
// ===== library types =====

TYPE "UDT_STRUCTANYPTR"
TITLE = 'DISSASEMBLED ANYPOINTER'
   STRUCT
      S7Code : Byte;
      DataType : Byte;
      Length : Int;
      DBNumber : Int;
      MemoryArea : Byte;
      ByteAddressMSB : Byte;
      ByteAddressLSB : Word;
   END_STRUCT;
END_TYPE

// ===== library: MasterCopy "Unixtime" =====

FUNCTION "Unixtime" : Void   // FC114, SCL
{ S7_Optimized_Access := 'FALSE' }
VERSION : 0.1
// ported by Groschke to TIA V13
BEGIN
   #leapyears := 0;
   #days_from_1970 := 0;

   // days of current month without leap day

   #days_from_BeginOfYear[0] := 0;
   #days_from_BeginOfYear[1] := 31;
   #days_from_BeginOfYear[2] := 59;
   #days_from_BeginOfYear[3] := 90;
   #days_from_BeginOfYear[4] := 120;
   #days_from_BeginOfYear[5] := 151;
   #days_from_BeginOfYear[6] := 181;
   #days_from_BeginOfYear[7] := 212;
   #days_from_BeginOfYear[8] := 243;
   #days_from_BeginOfYear[9] := 273;
   #days_from_BeginOfYear[10] := 304;
   #days_from_BeginOfYear[11] := 334;


   // read system time
   #sfc1_ret_val := RD_SYS_T(OUT => #CDT_systemtime);
   #year := BCD16_TO_INT(#systemtime.year_CDT) + 2000;
   #month := BCD16_TO_INT(#systemtime.month_CDT);
   #day := BCD16_TO_INT(#systemtime.day_CDT);
   #hour := BCD16_TO_INT(#systemtime.hour_CDT);
   #minute := BCD16_TO_INT(#systemtime.minute_CDT);
   #second := BCD16_TO_INT(#systemtime.second_CDT);


   // sum of leap years since 1979 (without current leap year)
   #leapyears := ((#year - 1) - 1968) / 4
   - ((#year - 1) - 1900) / 100
   + ((#year - 1) - 1600) / 400;


   #days_from_1970 := (#year - 1970) * 365 + #leapyears
   + #days_from_BeginOfYear[#month] + #day - 1;

   IF ((#month > 2) AND ((#year MOD 4 = 0) AND ((#year MOD 100 <> 0) OR (#year MOD 400 = 0)))) THEN
       #days_from_1970 := #days_from_1970 + 1; // + leap day, if year is leap year
   END_IF;

   // OUTPUT in s
   #l_unixtime := #second + 60 * (#minute + 60 * (#hour + 24 * #days_from_1970));


   // if error return 0
   IF #sfc1_ret_val <> 0 THEN
       #Unixtime := 0;
   ELSE
       #Unixtime := DINT_TO_DWORD(#l_unixtime);
   END_IF;
END_FUNCTION

// ===== library: MasterCopy "mqttExample" =====

FUNCTION_BLOCK "mqttExample"   // FB70, SCL
TITLE = 'MQTT Example Application'
{ S7_Optimized_Access := 'FALSE' }
AUTHOR : Brand
VERSION : 1.0
BEGIN
END_FUNCTION_BLOCK

// ===== library: MasterCopy "mqttRuntime" =====

FUNCTION_BLOCK "mqttRuntime"   // FB102, SCL
TITLE = 'Runtimercounter'
{ S7_Optimized_Access := 'FALSE' }
AUTHOR : Groschke
VERSION : 1.0
// ported by Groschke to TIA V13
BEGIN

   IF #IN AND NOT #FP_IN THEN
     #last := 0;
     #FP_IN := true;
   END_IF;

   IF NOT #IN AND #FP_IN THEN
     #FP_IN := false;
   END_IF;


   IF #IN AND NOT #RES THEN
     #now := DWORD_TO_DINT("Unixtime"());
     IF #last = 0 THEN
       #last := #now;
       GOTO Out;
     ELSE
       #run := #run + (#now - #last);
       #last := #now;
     END_IF;

   END_IF;

   IF #IN AND #RES THEN
     #run := 0;
     #now := 0;
     #last := 0;
   ELSIF NOT #IN AND #RES THEN
     #run := 0;
     #now := 0;
     #last := 0;
   END_IF;

   IF #run >= 2073600 THEN // avoid overflow of time typ 
     #run := 0;
   END_IF;

   Out:
   #RTIME := DINT_TO_TIME(#run * 1000);
END_FUNCTION_BLOCK

// ===== library: MasterCopy "mqttGlobals" =====

DATA_BLOCK "mqttGlobals"   // DB111
TITLE = 'MQTT CONSTANTS'
{ S7_Optimized_Access := 'FALSE' }
AUTHOR : Brand
VERSION : 0.1
   VAR
      MQTT_KEEPALIVE : Time;
      MQTT_SOCKET_TIMEOUT : Time;
      TCP_RECVBUFFERSIZE : Int;
      TCP_MAXRECVSIZE : Int;
      TCP_SENDBUFFERSIZE : Int;
      TCP_TIMEOUT : Time;
      MQTT_STATE_DISCONNECT : Int;
      MQTT_STATE_DISCONNECTING : Int;
      MQTT_CONNECTION_TIMEOUT : Int;
      MQTT_CONNECTION_LOST : Int;
      MQTT_CONNECT_FAILED : Int;
      MQTT_DISCONNECTED : Int;
      MQTT_CONNECTING : Int;
      MQTT_CONNECTED : Int;
      MQTT_CONN_ACCEPTED : Int;
      MQTT_CONN_BAD_PROTOCOL : Int;
      MQTT_CONN_BAD_CLIENT_ID : Int;
      MQTT_CONN_SRVUNAVAIL : Int;
      MQTT_CONN_BAD_CREDEN : Int;
      MQTT_CONN_UNAUTHORIZED : Int;
      MQTTCONNECT : Int;
      MQTTCONNACK : Int;
      MQTTPUBLISH : Int;
      MQTTPUBACK : Int;
      MQTTPUBREC : Int;
      MQTTPUBREL : Int;
      MQTTPUBCOMP : Int;
      MQTTSUBSCRIBE : Int;
      MQTTSUBACK : Int;
      MQTTUNSUBSCRIBE : Int;
      MQTTUNSUBACK : Int;
      MQTTPINGREQ : Int;
      MQTTPINGRESP : Int;
      MQTTDISCONNECT : Int;
      MQTTReserved : Int;
      MQTTQOS0 : Int;
      MQTTQOS1 : Int;
      MQTTQOS2 : Int;
   END_VAR
BEGIN
END_DATA_BLOCK

// ===== library: MasterCopy "mqttGetNextMessageID" =====

FUNCTION "mqttGetNextMessageID" : Void   // FC103, SCL
TITLE = 'MQTT Message ID Generator'
{ S7_Optimized_Access := 'FALSE' }
AUTHOR : Brand
VERSION : 1.0
BEGIN
     "mqttData".nextMsgId := "mqttData".nextMsgId + 1;

     IF ("mqttData".nextMsgId <= 0) THEN
       "mqttData".nextMsgId := 1;
     END_IF;

     #mqttGetNextMessageID := "mqttData".nextMsgId;
END_FUNCTION

// ===== library: MasterCopy "mqttCONNECT" =====

FUNCTION "mqttCONNECT" : Void   // FC101, SCL
TITLE = 'MQTT Connect Function'
{ S7_Optimized_Access := 'FALSE' }
AUTHOR : Brand
VERSION : 1.0
// ported by Groschke to TIA V13
BEGIN
END_FUNCTION

// ===== library: MasterCopy "mqttSimpleCONNECT" =====

FUNCTION "mqttSimpleCONNECT" : Void   // FC109, SCL
TITLE = 'MQTT Connect Function (basic parameters)'
{ S7_Optimized_Access := 'FALSE' }
AUTHOR : Brand
VERSION : 1.0
// ported by Groschke to TIA V13
BEGIN
     #l_clientID := #clientID;
     #l_cleanSession := #cleanSession;

     "mqttCONNECT"(clientID := #l_clientID,
                   withUsername := false,
                   withPassword := false,
                   cleanSession := #l_cleanSession,
                   withWill := false,
                   willQos := 0,
                   willRetain := 0,
                   willTopic := '',
                   willPayload := NULL,
                   willPayloadLength := 0,
                   username := '',
                   password := '');
END_FUNCTION

// ===== library: MasterCopy "mqttDISCONNECT" =====

FUNCTION "mqttDISCONNECT" : Void   // FC102, SCL
TITLE = 'MQTT Disconnect Function'
{ S7_Optimized_Access := 'FALSE' }
AUTHOR : Brand
VERSION : 1.0
// ported by Groschke to TIA V13
BEGIN
     "mqttData".buffer[0] := INT_TO_BYTE("mqttGlobals".MQTTDISCONNECT);
     "mqttData".buffer[1] := 0;
     "mqttSendTCP"(offset := 0,
                   size := 2);
     "mqttData".lastOutActivity := "mqttData".runTime;
     "mqttData"._state := "mqttGlobals".MQTT_DISCONNECTED;
END_FUNCTION

// ===== library: MasterCopy "mqttSUBSCRIBE" =====

FUNCTION "mqttSUBSCRIBE" : Void   // FC110, SCL
TITLE = 'MQTT Subscribe Function'
{ S7_Optimized_Access := 'FALSE' }
AUTHOR : Brand
VERSION : 1.0
// ported by Groschke to TIA V13
BEGIN

   // if there's no MQTT connection return
   IF "mqttData"._state = "mqttGlobals".MQTT_DISCONNECTED THEN
     RETURN;
   END_IF;

   #l_topic := #topic;

   // check if topic is not longer than 119 bytes
   IF (128 < (9 + LEN(#l_topic))) THEN
     RETURN;
   END_IF;

   #length := 5;

   // set message ID
   #thisMessageID := "mqttGetNextMessageID"();
   "mqttData".buffer[#length] := DWORD_TO_BYTE(SHR(IN := INT_TO_DWORD(#thisMessageID), N := 8));
   #length := #length + 1;
   "mqttData".buffer[#length] := INT_TO_BYTE(#thisMessageID) AND B#16#FF;
   #length := #length + 1;

   // set topic                
   #length := "mqttWriteString"(str := #l_topic, pos := #length);

   // set topic qos
   "mqttData".buffer[#length] := INT_TO_BYTE(#topicQos);
   #length := #length + 1;

   // write header and send message
   "mqttWrite"(header := INT_TO_BYTE("mqttGlobals".MQTTSUBSCRIBE),
               length := #length - 5);
END_FUNCTION

// ===== library: MasterCopy "mqttUNSUBSCRIBE" =====

FUNCTION "mqttUNSUBSCRIBE" : Void   // FC111, SCL
TITLE = 'MQTT Unsubscribe Function'
{ S7_Optimized_Access := 'FALSE' }
AUTHOR : Brand
VERSION : 1.0
BEGIN

   // if there's no MQTT connection return
   IF "mqttData"._state = "mqttGlobals".MQTT_DISCONNECTED THEN
     RETURN;
   END_IF;

   #l_topic := #topic;

   // check if topic is not longer than 119 bytes
   IF (128 < (9 + LEN(#l_topic))) THEN
     RETURN;
   END_IF;

   #length := 5;

   // set message ID
   #thisMessageID := "mqttGetNextMessageID"();
   "mqttData".buffer[#length] := DWORD_TO_BYTE(SHR(IN := INT_TO_DWORD(#thisMessageID), N := 8));
   #length := #length + 1;
   "mqttData".buffer[#length] := INT_TO_BYTE(#thisMessageID) AND B#16#FF;
   #length := #length + 1;

   // set topic        
   #length := "mqttWriteString"(str := #l_topic, pos := #length);

   #fixedHeader := INT_TO_BYTE("mqttGlobals".MQTTUNSUBSCRIBE);
   // Set Header Flags for duplicates, qos level and retain
   #fixedHeader := #fixedHeader OR SHL(IN := BOOL_TO_BYTE(true), N := 1);

   // write header and send message
   "mqttWrite"(header := #fixedHeader,
               length := #length - 5);
END_FUNCTION

// ===== library: MasterCopy "mqttPUBLISH" =====

FUNCTION "mqttPUBLISH" : Void   // FC105, SCL
TITLE = MQTT Publish Function
{ S7_Optimized_Access := 'FALSE' }
AUTHOR : Brand
VERSION : 1.0
// ported by Groschke to TIA V13
BEGIN
   // set return value (message ID) to 0
   #mqttPUBLISH := 0;

   // if there's no MQTT connection return an error code
   IF "mqttData"._state = "mqttGlobals".MQTT_DISCONNECTED THEN
     #mqttPUBLISH := -1;
     RETURN;
   END_IF;

   // Fixed header, byte 1
   // +--------+---+-----+---+---+----------+-----+-----+--------+
   // |bit     | 7 |  6  | 5 | 4 |     3    |  2  |  1  |    0   |
   // +--------+---+-----+---+---+----------+-----+-----+--------+
   // |byte 1  | Message Type(3) | DUP Flag | QoS level | RETAIN |
   // +--------+-----------------+----------+-----------+--------+

   // set package type in header
   #fixedHeader := INT_TO_BYTE("mqttGlobals".MQTTPUBLISH);
   // Set Header Flags for duplicates, qos level and retain
   #fixedHeader := #fixedHeader OR SHL(IN := BOOL_TO_BYTE(#duplicate), N := 3) OR SHL(IN := INT_TO_BYTE(#qos), N := 1) OR BOOL_TO_BYTE(#retain);

   // Fixed header, byte 2
   // +--------+---+---+---+---+---+---+---+---+
   // |bit     | 7 | 6 | 5 | 4 | 3 | 2 | 1 | 0 |
   // +--------+---+---+---+---+---+---+---+---+
   // |bytes 2..4|   Remaining Length          |
   // +--------+-------------------------------+

   // Variable header, topic
   // +--------+---+---+---+---+---+---+---+---+
   // |bit     | 7 | 6 | 5 | 4 | 3 | 2 | 1 | 0 |
   // +--------+---+---+---+---+---+---+---+---+
   // |byte    |           Topic length MSB    |
   // +~~~~~~~~|~~~~~~~~~~~~~~~~~~~~~~~~~~~~~~~+
   // |byte    |           Topic length LSB    |
   // +~~~~~~~~|~~~~~~~~~~~~~~~~~~~~~~~~~~~~~~~+
   // +--------+---+---+---+---+---+---+---+---+
   // |bit     | 7 | 6 | 5 | 4 | 3 | 2 | 1 | 0 |
   // +--------+---+---+---+---+---+---+---+---+
   // |bytes    |           Topic              |
   // +~~~~~~~~|~~~~~~~~~~~~~~~~~~~~~~~~~~~~~~~+

   // point to buffer area in front of fixed header (5 bytes)
   // copy topic to buffer
   #holdstring := #topic;
   #length := 5;

   #length := "mqttWriteString"(str := #holdstring, pos := #length);

   // MessageID  
   // Variable header, byte 9
   // +--------+---+---+---+---+---+---+---+---+
   // |bit     | 7 | 6 | 5 | 4 | 3 | 2 | 1 | 0 |
   // +--------+---+---+---+---+---+---+---+---+           
   // |byte    |       Message ID LSB (0)      |
   // +--------+-------------------------------+ 
   // |byte    |       Message ID LSB (10)     |
   // +--------+-------------------------------+

   // set MessageID if qos level 1 or 2
   IF (#qos = "mqttGlobals".MQTTQOS1) OR (#qos = "mqttGlobals".MQTTQOS2) THEN
     IF #messageid > 0 THEN
       #thisMessageID := #messageid;
     ELSE
       #thisMessageID := "mqttGetNextMessageID"();
     END_IF;

     // insert message ID
     "mqttData".buffer[#length] := DWORD_TO_BYTE(SHR(IN := INT_TO_DWORD(#thisMessageID), N := 8));
     #length := #length + 1;
     "mqttData".buffer[#length] := INT_TO_BYTE(#thisMessageID) AND B#16#FF;
     #length := #length + 1;

     #mqttPUBLISH := #thisMessageID;
   END_IF;

   // Payload
   // Variable header, byte 11...
   // +--------+---+---+---+---+---+---+---+---+
   // |bit     | 7 | 6 | 5 | 4 | 3 | 2 | 1 | 0 |
   // +--------+---+---+---+---+---+---+---+---+           
   // |bytes   |           Payload             |
   // +~~~~~~~~|~~~~~~~~~~~~~~~~~~~~~~~~~~~~~~~+  

   // copy payload to buffer
   //ptrBuffer := mqttData.buffer[length];
   #ptrPayload := #payload;

   IF #payloadLength > 0 THEN
     FOR #i := 0 TO #payloadLength - 1 DO
       #ret := BLKMOV(SRCBLK := #ptrPayload, DSTBLK => "mqttData".buffer[#length]);
       // what is this?!
       IF #ret <> 0 THEN
         //m23.2 := true;
         //return
         ;
       END_IF;
       #length := #length + 1;
       #structPtrPayload.ByteAddressLSB := INT_TO_WORD(WORD_TO_INT(#structPtrPayload.ByteAddressLSB) + 8);
     END_FOR;
   END_IF;

   // copy header information (includes remaining length calculation)
   // and trigger tcpsend
   "mqttWrite"(header := #fixedHeader,
               length := #length - 5);
END_FUNCTION

// ===== library: MasterCopy "mqttPUBACK" =====

FUNCTION "mqttPUBACK" : Void   // FC104, SCL
TITLE = 'MQTT Publish Acknowledge QoS1 Function'
{ S7_Optimized_Access := 'FALSE' }
AUTHOR : Brand
VERSION : 1.0
BEGIN
     "mqttData".buffer[0] := INT_TO_BYTE("mqttGlobals".MQTTPUBACK);
     "mqttData".buffer[1] := 2;
     "mqttData".buffer[2] := #packetIdMSB;
     "mqttData".buffer[3] := #packetIdLSB;
     "mqttSendTCP"(offset := 0,
                   size := 4);
     "mqttData".lastOutActivity := "mqttData".runTime;
END_FUNCTION

// ===== library: MasterCopy "mqttSendTCP" =====

FUNCTION "mqttSendTCP" : Void   // FC108, SCL
TITLE = 'MQTT mqttSendTCP Helper Function'
{ S7_Optimized_Access := 'FALSE' }
AUTHOR : Brand
VERSION : 1.0
// ported by Groschke to TIA V13
BEGIN
   IF "mqttData".sendSize + #size <= "mqttGlobals".TCP_SENDBUFFERSIZE THEN
     FOR #i := 0 TO #size - 1 DO
       "mqttData".tcpSendBuf[MIN(IN1 := (#i + "mqttData".sendSize), IN2 := "mqttGlobals".TCP_SENDBUFFERSIZE)] := "mqttData".buffer[#offset + #i];
     END_FOR;
     "mqttData".sendSize := "mqttData".sendSize + #size;
     "mqttData".reqSend := true;
   ELSE
     "mqttData".tcp_sendBufferFull := true;
   END_IF;
END_FUNCTION

// ===== library: MasterCopy "mqttWrite" =====

FUNCTION "mqttWrite" : Void   // FC112, SCL
TITLE = 'MQTT mqttWrite Helper Function'
{ S7_Optimized_Access := 'FALSE' }
AUTHOR : Brand
VERSION : 1.0
// ported by Groschke to TIA V13
BEGIN
   #llen := 0;
   #pos := 0;
   #_len := #length;
   REPEAT
     #digit := INT_TO_BYTE(#_len MOD 128);
     #_len := #_len / 128;
     IF (#_len > 0) THEN
       #digit_bitview[7] := 1; // digit |= 0x80;
     END_IF;
     #lenBuf[#pos] := #digit;
     #pos := #pos + 1;
     #llen := #llen + 1;
   UNTIL (#_len <= 0) // do..while(len>0)
   END_REPEAT;
   "mqttData".buffer[4 - #llen] := #header;
   FOR #i := 0 TO #llen - 1 DO
     "mqttData".buffer[5 - #llen + #i] := #lenBuf[#i];
   END_FOR;
   "mqttSendTCP"(offset := 4 - #llen,
                 size := #length + 1 + #llen);
   "mqttData".lastOutActivity := "mqttData".runTime;
END_FUNCTION

// ===== library: MasterCopy "mqttWriteString" =====

FUNCTION "mqttWriteString" : Void   // FC113, SCL
TITLE = MQTT mqttWriteString Helper Function
{ S7_Optimized_Access := 'FALSE' }
AUTHOR : Brand
VERSION : 1.0
// ported by Groschke to TIA V13
BEGIN
   #newPos := #pos + 2;
   #i := 0;

   FOR #j := 1 TO BYTE_TO_INT(#_str.act_length) DO
     "mqttData".buffer[#newPos] := #_str.str[#j];
     #newPos := #newPos + 1;
     #i := #i + 1;
   END_FOR;

   "mqttData".buffer[#newPos - 2 - #i] := DWORD_TO_BYTE(SHR(IN := DINT_TO_DWORD(#i), N := 8));
   "mqttData".buffer[#newPos - 1 - #i] := DINT_TO_BYTE(#i);

   #mqttWriteString := #newPos;
END_FUNCTION

// ===== library: MasterCopy "mqttAvailable" =====

FUNCTION "mqttAvailable" : Void   // FC100, SCL
TITLE = 'MQTT mqttAvailable Helper Function'
{ S7_Optimized_Access := 'FALSE' }
AUTHOR : Brand
VERSION : 1.0
BEGIN
   #mqttAvailable := ("mqttData".pRead <> "mqttData".pRec) OR "mqttData".RecBufFull;
END_FUNCTION

// ===== library: MasterCopy "mqttReadByte" =====

FUNCTION "mqttReadByte" : Void   // FC106, SCL
TITLE = 'MQTT mqttReadByte Helper Function'
{ S7_Optimized_Access := 'FALSE' }
AUTHOR : Brand
VERSION : 1.0
BEGIN
   #mqttReadByte := "mqttData".tcpRecBuf["mqttData".pRead];
   "mqttData".pRead := "mqttData".pRead + 1;
   IF ("mqttData".pRead >= "mqttGlobals".TCP_RECVBUFFERSIZE) THEN
     "mqttData".pRead := 0;
   END_IF;
   "mqttData".RecBufFull := false;
END_FUNCTION

// ===== library: MasterCopy "mqttReadByteToBuf" =====

FUNCTION "mqttReadByteToBuf" : Void   // FC107, SCL
TITLE = 'MQTT mqttReadByteToBuf Helper Function'
{ S7_Optimized_Access := 'FALSE' }
AUTHOR : Brand
VERSION : 1.0
BEGIN
   #cur_index := #pos;
   #readed := "mqttReadByte"();
   "mqttData".buffer[#cur_index] := #readed;
   #cur_index := #cur_index + 1;
   #mqttReadByteToBuf := #cur_index;
END_FUNCTION

// ===== library: MasterCopy "mqttPacketReader" =====

FUNCTION_BLOCK "mqttPacketReader"   // FB101, SCL
TITLE = 'MQTT mqttPacketReader Helper Function'
{ S7_Optimized_Access := 'FALSE' }
AUTHOR : Brand
VERSION : 1.0
BEGIN
   CASE (#State) OF
     -1: // Alternative to original blocking call
       IF (("mqttData".runTime - #previousTime) >= "mqttGlobals".MQTT_SOCKET_TIMEOUT) THEN
         #xDone := true;
         #result := 0;
         #State := 0;
       ELSIF "mqttAvailable"() THEN
         #State := #oldState;
       END_IF;
     0: // Wait for Start
       #oldState := 0;
       IF (#iBegin) THEN
         #iBegin := false;
         #xDone := false;
         #_len := 0;
         #State := 1;
       END_IF;
     1:    // Getting first byte
       #oldState := 1;
       IF "mqttAvailable"() THEN
         #_len := "mqttReadByteToBuf"(pos := #_len);
         #isPublish := BYTE_TO_INT("mqttData".buffer[0] AND B#16#F0) = "mqttGlobals".MQTTPUBLISH;
         #multiplier := 1;
         #length := 0;
         #digit := B#16#00;
         #start := 0;
         #State := 2;
       ELSE
         #previousTime := "mqttData".runTime;
         #State := -1;
       END_IF;
     2: // do..while((digit & 128) != 0) loop equivalent
       #oldState := 2;
       IF "mqttAvailable"() THEN
         #digit := "mqttReadByte"();
         "mqttData".buffer[#_len] := #digit;
         #_len := #_len + 1;
         #length := #length + (BYTE_TO_DINT(#digit AND B#16#7F) * #multiplier);
         #multiplier := #multiplier * 128;
         IF (#digit AND B#16#80) = B#16#00 THEN
           #lengthLength := #_len - 1;
           IF (#isPublish) THEN
             #State := 3;
           ELSE
             #State := 5;
           END_IF;
         END_IF;
       ELSE
         #previousTime := "mqttData".runTime;
         #State := -1;
       END_IF;
     3:    // First Publish Byte
       #oldState := 3;
       IF "mqttAvailable"() THEN
         #_len := "mqttReadByteToBuf"(pos := #_len);
         #State := 4;
       ELSE
         #previousTime := "mqttData".runTime;
         #State := -1;
       END_IF;
     4:    // Second Publish Byte
       #oldState := 4;
       IF "mqttAvailable"() THEN
         #_len := "mqttReadByteToBuf"(pos := #_len);
         #start := 2;
         #State := 5;
       ELSE
         #previousTime := "mqttData".runTime;
         #State := -1;
       END_IF;
     5:    // Read rest of Packet (for loop replacement)
       #oldState := 5;
       //loop exit
       IF (#start = #length) THEN
         IF (#_len > "mqttGlobals".TCP_MAXRECVSIZE) THEN
           #_len := 0; // just drop packet if too long
         END_IF;
         #xDone := true;
         #result := #_len;
         #State := 0;
       ELSIF "mqttAvailable"() THEN
         #digit := "mqttReadByte"();
         IF (#_len < "mqttGlobals".TCP_MAXRECVSIZE) THEN
           "mqttData".buffer[#_len] := #digit;
         END_IF;
         #_len := #_len + 1;
         //loop
         #start := #start + 1;
       ELSE
         #previousTime := "mqttData".runTime;
         #State := -1;
       END_IF;
   END_CASE;
END_FUNCTION_BLOCK

// ===== library: MasterCopy "mqttData" =====

DATA_BLOCK "mqttData"   // DB1
TITLE = 'MQTT DATABLOCK'
{ S7_Optimized_Access := 'FALSE' }
AUTHOR : Brand
VERSION : 0.1
   VAR
      tcpRecBuf : Array[0..8192] of Byte;
      pRec : Int;
      pRead : Int;
      RecBufFull : Bool;
      tcpSendBuf : Array[0..4096] of Byte;
      reqSend : Bool;
      sendSize : Int;
      buffer : Array[0..4096] of Byte;
      nextMsgId : Int;
      _state : Int;
      packet_state : Int;
      pingOutstanding : Bool;
      lastInActivity : Time;
      lastOutActivity : Time;
      runTime : Time;
      ethTCPConnected : Bool;
      mqttErrorCode : Int;
      recPublishPacketID : Int;
      tcp_sendBufferFull : Bool;
   END_VAR
BEGIN
END_DATA_BLOCK

// ===== library: MasterCopy "MQTT" =====

FUNCTION_BLOCK "MQTT"   // FB100, SCL
TITLE = 'MQTT MAIN Function(PN)'
{ S7_Optimized_Access := 'FALSE' }
AUTHOR : Maul
VERSION : 1.0
BEGIN
END_FUNCTION_BLOCK